{attribute addProperty BoxType "EJ1957-0000-0017"}
{attribute addProperty Id "Module_1_FSOEModule_1_FSOE_B52BB714112140Module_2_FSOUTModule_2_FSOUT_B889B7D03240Module_3_DEVICEIOModule_3_DEVICEIO_FB2B67D71620Module_4_FSLOGICModule_4_FSLOGIC_3E6251391620WcStateAT %I*WcState_DC9C971540.50InfoDataAT %I*InfoData_BC63D37F80100"}
{attribute addProperty CRC "2859848888"}
{attribute addProperty SizeInBites "260"}
{attribute addProperty SizeInBytes "32.5"}
TYPE EJ1957_6B6926D1 :
STRUCT
	{attribute addProperty Name "Module_1_FSOE"}
	Module_1_FSOE : Module_1_FSOE_B52BB714;
	{attribute addProperty Name "Module_2_FSOUT"}
	Module_2_FSOUT : Module_2_FSOUT_B889B7D0;
	{attribute addProperty Name "Module_3_DEVICEIO"}
	Module_3_DEVICEIO : Module_3_DEVICEIO_FB2B67D7;
	{attribute addProperty Name "Module_4_FSLOGIC"}
	Module_4_FSLOGIC : Module_4_FSLOGIC_3E625139;
	{attribute addProperty Name "WcState"}
	WcState : WcState_DC9C9715;
	{attribute addProperty Name "InfoData"}
	InfoData : InfoData_BC63D37F;
END_STRUCT
END_TYPE

(* stored: Version 1.2.0.0, ProductVersion 3.1.4024.9
   DUT EJ1957_6B6926D1: Id {1c147236-6c3a-445e-9767-9a56fd93b4e5} *)
